{attribute 'qualified_only'}
VAR_GLOBAL
	// Raw data read every cycle
	gl_voltage_effective_raw AT %I* : INT := 15000;
	gl_voltage_periode_raw AT  %I* : UINT := 20;
	gl_current_effective_raw AT %I* : INT := 3800;
	gl_current_periode_raw AT %I* : UINT := 20;
END_VAR

(* stored: Version 1.1.0.1, ProductVersion 3.1.4024.12
   GVL GVL: Id {71bba7d0-3505-4f0b-8492-903f27a2e840} *)
